// TIA Portal V19 export
FUNCTION_BLOCK "TYPIC_C501_IF_BBI"   // FB5, FBD
TITLE = TYPIC_C501_IF_BBI: Brandblusinstallatie
{ S7_Optimized_Access := 'TRUE' }
AUTHOR : OCOTECH
FAMILY : Typical
NAME : C501.701
// Logisch Object Besturing: C501.701
// 
// De interne functie brandblusinstallatie verwerkt de algemene bedieningen vanop het aanraakscherm en de algemene sturingen van de brandblusinstallatie.
// stored: MemoryReserve 10, SetENOAutomatically false
   VAR_INPUT
      EXT_HW { ExternalAccessible := 'False'; ExternalVisible := 'False'; ExternalWritable := 'False'} : Bool;   // Sturings hardware (PLC) bewaking (1 = OK)
      IN_STS1 { ExternalAccessible := 'False'; ExternalVisible := 'False'; ExternalWritable := 'False'} : Bool;   // Status schuif ALSB ingeschakeld
      IN_STS2 { ExternalAccessible := 'False'; ExternalVisible := 'False'; ExternalWritable := 'False'} : Bool;   // Status schuif ALSB in test
      IN_STS3 { ExternalAccessible := 'False'; ExternalVisible := 'False'; ExternalWritable := 'False'} : Bool;   // Status schuif ALSB uitgereden
      IN_AUT { ExternalAccessible := 'False'; ExternalVisible := 'False'; ExternalWritable := 'False'} : Bool;   // Beveiliging in ALSB-bord (1 = OK)
      IN_NB_AUT { ExternalAccessible := 'False'; ExternalVisible := 'False'; ExternalWritable := 'False'} : Bool;   // Beveiliging No-Break (1 = OK)
      IN_SPD_OK { ExternalAccessible := 'False'; ExternalVisible := 'False'; ExternalWritable := 'False'} : Bool;   // Status overspanningsbeveiliging (1 = OK)
      IN_KST_AUT { ExternalAccessible := 'False'; ExternalVisible := 'False'; ExternalWritable := 'False'} : Bool;   // Beveiliging kastklimatisatie (1 = OK)
      IN_KST_AAN { ExternalAccessible := 'False'; ExternalVisible := 'False'; ExternalWritable := 'False'} : Bool;   // Lastscheider aan (1 = AAN)
      IN_LDE { ExternalAccessible := 'False'; ExternalVisible := 'False'; ExternalWritable := 'False'} : Bool;   // Lekdetectie in pomplokaal (1 = OK)
   END_VAR
   VAR_OUTPUT
      VAR_IF_BBI { ExternalAccessible := 'False'; ExternalVisible := 'False'; ExternalWritable := 'False'} : "C501_VAR_IF_BBI_TYPIC";   // Struct met alle variabelen naar de basisfunctie
   END_VAR
   VAR_IN_OUT
      STU_IF_BBI : "C501_STU_IF_BBI_TYPIC";   // Struct met alle sturingen vanuit de basisfunctie
   END_VAR
   VAR
      BED : Struct   // Bedieningen
         UIT : Bool;   // Bediening om regime Uit te activeren
         BWK : Bool;   // Bediening om regime Bewaken te activeren
         BLUS1 : Bool;   // Bediening om regime Blussen Hydrant te activeren
         BLUS2 : Bool;   // Bediening om regime Blussen Hydrant en WMS te activeren
         TEST : Bool;   // Bediening om regime Testen te activeren
      END_STRUCT;
      STO { ExternalWritable := 'False'} : Struct   // Storingen
         A001 : Bool;   // Beveiliging aangesproken
         A002 : Bool;   // Beveiliging No-Break aangesproken
         A003 : Bool;   // Schuif ALSB uitgeschakeld
         A004 : Bool;   // Schuif ALSB in test
         A005 : Bool;   // Schuif ALSB uitgereden
         A006 : Bool;   // Lekdetectie in pomplokaal
         A007 : Bool;   // Overspanningsbeveiliging aangesproken
         A008 : Bool;   // Beveiliging kastklimatisatie aangesproken
         A009 : Bool;   // Lastscheider niet aan
      END_STRUCT;
      VAR { ExternalWritable := 'False'} : Struct   // Variabelen
         WRE : USInt;   // Actueel actief regime
         REQ_UIT { ExternalAccessible := 'False'; ExternalVisible := 'False'} : Bool;   // Aanvraag om regime Uit te activeren
         REQ_BWK { ExternalAccessible := 'False'; ExternalVisible := 'False'} : Bool;   // Aanvraag om regime Bewaken te activeren
         REQ_BLUS1 { ExternalAccessible := 'False'; ExternalVisible := 'False'} : Bool;   // Aanvraag om regime Blussen Hydrant te activeren
         REQ_BLUS2 { ExternalAccessible := 'False'; ExternalVisible := 'False'} : Bool;   // Aanvraag om regime Blussen Hydrant en WMS te activeren
         REQ_TEST { ExternalAccessible := 'False'; ExternalVisible := 'False'} : Bool;   // Aanvraag om regime Testen te activeren
         EXT_HW { ExternalAccessible := 'False'; ExternalVisible := 'False'} : Bool;   // Sturings hardware (PLC) in storing
      END_STRUCT;
   END_VAR
BEGIN

REGION Network 1: START
END_REGION

REGION Network 2: +++ Bedieningen +++
   // Verwerking van de bedieningen.
END_REGION

REGION Network 3: +++ Storingen +++
   // Verwerken van de storingsmeldingen.
END_REGION

REGION Network 4: Storing A001: Beveiliging aangesproken
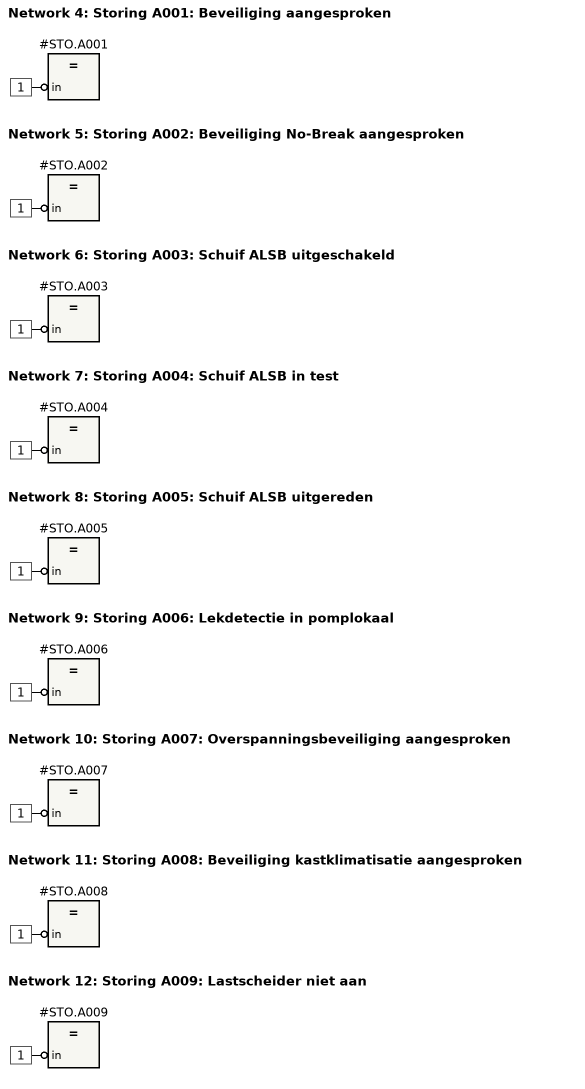
   #STO.A001 := NOT 1;
END_REGION

REGION Network 5: Storing A002: Beveiliging No-Break aangesproken
   #STO.A002 := NOT 1;
END_REGION

REGION Network 6: Storing A003: Schuif ALSB uitgeschakeld
   #STO.A003 := NOT 1;
END_REGION

REGION Network 7: Storing A004: Schuif ALSB in test
   #STO.A004 := NOT 1;
END_REGION

REGION Network 8: Storing A005: Schuif ALSB uitgereden
   #STO.A005 := NOT 1;
END_REGION

REGION Network 9: Storing A006: Lekdetectie in pomplokaal
   #STO.A006 := NOT 1;
END_REGION

REGION Network 10: Storing A007: Overspanningsbeveiliging aangesproken
   #STO.A007 := NOT 1;
END_REGION

REGION Network 11: Storing A008: Beveiliging kastklimatisatie aangesproken
   #STO.A008 := NOT 1;
END_REGION

REGION Network 12: Storing A009: Lastscheider niet aan
   #STO.A009 := NOT 1;
END_REGION

REGION Network 13: +++ Actieve werkingsregime aangeven +++
   // Het actieve werkingsregime wordt ontvangen vanuit de basisfunctie en wordt naar een interne variabele weggeschreven zodat het actieve werkingsregime kan aangegeven worden op het aanraakscherm.
END_REGION

REGION Network 14 (SCL): EINDE
   // Variabelen van intern scada rakvlak naar outputs copieren
   #VAR_IF_BBI.REQ_UIT := #VAR.REQ_UIT;
   #VAR_IF_BBI.REQ_BWK := #VAR.REQ_BWK;
   #VAR_IF_BBI.REQ_BLUS1 := #VAR.REQ_BLUS1;
   #VAR_IF_BBI.REQ_BLUS2 := #VAR.REQ_BLUS2;
   #VAR_IF_BBI.REQ_TEST := #VAR.REQ_TEST;
   #VAR_IF_BBI.EXT_HW := #VAR.EXT_HW;
   #VAR_IF_BBI.STO := #STO;
END_REGION
END_FUNCTION_BLOCK
